(* PLC project Python_3, Неизвестно Python 1 *)
(* stored: creationDateTime 2020-11-18T10:24:47, modificationDateTime 2020-11-18T10:55:59 *)

(* main *)
PROGRAM main
  VAR
    In : INT;
    Out : INT;
    b_Triger : BOOL := False;
    python_eval0 : python_eval;
  END_VAR
  VAR  (* added by the conversion: wires and edge detectors of the diagram *)
    _NOT2_OUT : BOOL;
  END_VAR

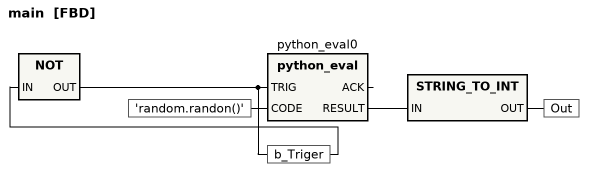
(* FBD diagram, written out as Structured Text *)
_NOT2_OUT := NOT b_Triger;
b_Triger := _NOT2_OUT;
python_eval0(TRIG := _NOT2_OUT, CODE := 'random.randon()');
Out := STRING_TO_INT(python_eval0.RESULT);
END_PROGRAM

CONFIGURATION config
  RESOURCE resource1 ON PLC
    TASK main_task(INTERVAL := T#1s0ms, PRIORITY := 0);
    PROGRAM maiin : main;
  END_RESOURCE
END_CONFIGURATION
